PROGRAM MAIN
VAR
	
	//Pulsador AT %I*: BOOL;
	//Lampara AT %Q*: BOOL;
	
	test_pieza: FB_Bloque;

END_VAR

test_pieza();

END_PROGRAM

(* stored: Version 1.1.0.1, ProductVersion 3.1.4024.12
   POU MAIN: Id {56f4075e-4895-4e88-bf82-4d98b9642bb1}, SpecialFunc None *)
